// TIA Portal project "practica 9" (V15)

(* hardware
DEVICE "S7-1200 station_1"  S7-1200 Station
   slot 0: "Rack_0"  S7-1200 Rack  Rack  V1.0
   slot 1: "PLC_1"  CPU 1214C AC/DC/Rly  6ES7 214-1BE30-0XB0  V2.2
   slot 3: "AQ 1x12BIT_1"  AQ1 signal board  6ES7 232-4HA30-0XB0  V1.0
DEVICE "S7-1200 station_2"  S7-1200 Station
   slot 0: "Rack_0"  S7-1200 Rack  Rack  V1.0
   slot 1: "PLC_2"  CPU 1214C AC/DC/Rly  6ES7 214-1BG40-0XB0  V4.2
DEVICE "HMI_1"  KTP700 Basic PN
   slot 0: "HMI_1"  KTP700 Basic PN  6AV2 123-2GB03-0AX0  15.0.0.0
   slot 1: "HMI_RT_1"  KTP700 Basic PN  6AV2 123-2GB03-0AX0  15.0.0.0
   slot 5: "HMI_1.IE_CP_1"  PROFINET Interface  15.0.0.0
      slot 1: "Interfaz PROFINET_1"  PROFINET Interface
         slot 1: "Port_1"  Port
*)

// ===== PLC "PLC_1"  CPU 1214C AC/DC/Rly =====

VAR_GLOBAL   // PLC tag table "Tabla de variables estándar"
   "PM" AT %I0.0 : Bool;
   "Paro" AT %I0.1 : Bool;
   "luz verde" AT %Q0.0 : Bool;
   "luz ambar" AT %Q0.1 : Bool;
   "luz roja" AT %Q0.2 : Bool;
   "bucle" AT %M5.0 : Bool;
   "Tag_1" AT %M5.1 : Bool;
   "Luz verde peaton" AT %Q0.4 : Bool;
   "Luz roja peaton" AT %Q0.5 : Bool;
   "Tag_2" AT %M5.2 : Bool;
   "Tag_3" AT %M5.3 : Bool;
END_VAR

// folder: System blocks/Program resources

DATA_BLOCK "IEC_Timer_0_DB"   // DB1
{ S7_Optimized_Access := 'TRUE' }
AUTHOR : Simatic
FAMILY : IEC
NAME : IEC_TMR
VERSION : 1.0
// stored: InstanceOfName IEC_TIMER
"IEC_TIMER"
BEGIN
END_DATA_BLOCK

DATA_BLOCK "IEC_Timer_0_DB_1"   // DB2
{ S7_Optimized_Access := 'TRUE' }
AUTHOR : Simatic
FAMILY : IEC
NAME : IEC_TMR
VERSION : 1.0
// stored: InstanceOfName IEC_TIMER
"IEC_TIMER"
BEGIN
END_DATA_BLOCK

DATA_BLOCK "IEC_Timer_0_DB_2"   // DB3
{ S7_Optimized_Access := 'TRUE' }
AUTHOR : Simatic
FAMILY : IEC
NAME : IEC_TMR
VERSION : 1.0
// stored: InstanceOfName IEC_TIMER
"IEC_TIMER"
BEGIN
END_DATA_BLOCK

DATA_BLOCK "IEC_Timer_0_DB_3"   // DB4
{ S7_Optimized_Access := 'TRUE' }
AUTHOR : Simatic
FAMILY : IEC
NAME : IEC_TMR
VERSION : 1.0
// stored: InstanceOfName IEC_TIMER
"IEC_TIMER"
BEGIN
END_DATA_BLOCK

DATA_BLOCK "IEC_Timer_0_DB_4"   // DB5
{ S7_Optimized_Access := 'TRUE' }
AUTHOR : Simatic
FAMILY : IEC
NAME : IEC_TMR
VERSION : 1.0
// stored: InstanceOfName IEC_TIMER
"IEC_TIMER"
BEGIN
END_DATA_BLOCK

DATA_BLOCK "IEC_Timer_0_DB_5"   // DB6
{ S7_Optimized_Access := 'TRUE' }
AUTHOR : Simatic
FAMILY : IEC
NAME : IEC_TMR
VERSION : 1.0
// stored: InstanceOfName IEC_TIMER
"IEC_TIMER"
BEGIN
END_DATA_BLOCK

DATA_BLOCK "IEC_Timer_0_DB_6"   // DB7
{ S7_Optimized_Access := 'TRUE' }
AUTHOR : Simatic
FAMILY : IEC
NAME : IEC_TMR
VERSION : 1.0
// stored: InstanceOfName IEC_TIMER
"IEC_TIMER"
BEGIN
END_DATA_BLOCK

// folder: (top level)

ORGANIZATION_BLOCK "Main"   // OB1, LAD, ProgramCycle
TITLE = "Main Program Sweep (Cycle)"
{ S7_Optimized_Access := 'TRUE' }
VERSION : 0.1
   VAR_TEMP   // added for the SCL form of the ladder/FBD networks
      _w1 : Bool;
      _w2 : Bool;
   END_VAR
BEGIN

REGION Network 1
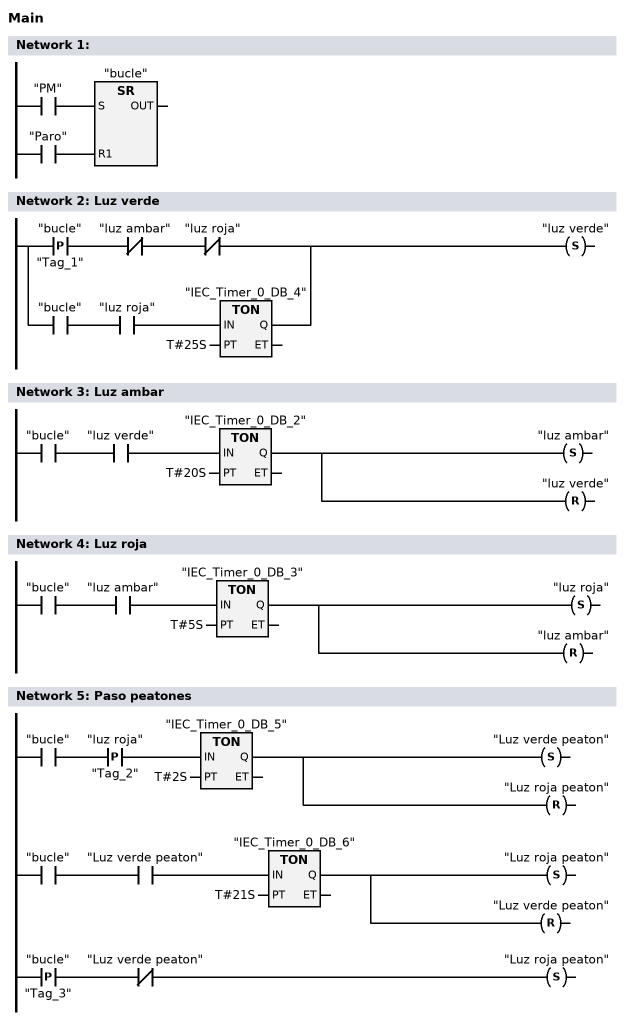
   RUNG wire#powerrail
      Contact( "PM" )
      S_SR(operand := "bucle", r1 := wire#w1)
   END_RUNG
   RUNG wire#powerrail
      Contact( "Paro" )
   END_RUNG wire#w1
   // the same network as SCL:
   IF "PM" THEN
       "bucle" := TRUE;   // SR flip-flop
   END_IF;
   IF "Paro" THEN "bucle" := FALSE; END_IF;
END_REGION

REGION Network 2: Luz verde
   #_w1 := "bucle" AND NOT "Tag_1";   // rising edge of "bucle"
   "Tag_1" := "bucle";
   "IEC_Timer_0_DB_4".TON(IN := "bucle" AND "luz roja", PT := T#25S);
   IF (#_w1 AND NOT "luz ambar" AND NOT "luz roja") OR "IEC_Timer_0_DB_4".Q THEN "luz verde" := TRUE; END_IF;
END_REGION

REGION Network 3: Luz ambar
   "IEC_Timer_0_DB_2".TON(IN := "bucle" AND "luz verde", PT := T#20S);
   IF "IEC_Timer_0_DB_2".Q THEN
       "luz ambar" := TRUE;
       "luz verde" := FALSE;
   END_IF;
END_REGION

REGION Network 4: Luz roja
   "IEC_Timer_0_DB_3".TON(IN := "bucle" AND "luz ambar", PT := T#5S);
   IF "IEC_Timer_0_DB_3".Q THEN
       "luz roja" := TRUE;
       "luz ambar" := FALSE;
   END_IF;
END_REGION

REGION Network 5: Paso peatones
   #_w1 := "bucle" AND "luz roja" AND NOT "Tag_2";   // rising edge of "luz roja"
   "Tag_2" := "luz roja";
   "IEC_Timer_0_DB_5".TON(IN := #_w1, PT := T#2S);
   IF "IEC_Timer_0_DB_5".Q THEN
       "Luz verde peaton" := TRUE;
       "Luz roja peaton" := FALSE;
   END_IF;
   "IEC_Timer_0_DB_6".TON(IN := "bucle" AND "Luz verde peaton", PT := T#21S);
   IF "IEC_Timer_0_DB_6".Q THEN
       "Luz roja peaton" := TRUE;
       "Luz verde peaton" := FALSE;
   END_IF;
   #_w2 := "bucle" AND NOT "Tag_3";   // rising edge of "bucle"
   "Tag_3" := "bucle";
   IF #_w2 AND NOT "Luz verde peaton" THEN "Luz roja peaton" := TRUE; END_IF;
END_REGION

REGION Network 6: Paro peaton
END_REGION
END_ORGANIZATION_BLOCK

// ===== PLC "PLC_2"  CPU 1214C AC/DC/Rly =====

VAR_GLOBAL   // PLC tag table "Tabla de variables estándar"
   "PM" AT %M5.5 : Bool;
   "Paro" AT %I0.1 : Bool;
   "luz verde" AT %Q0.0 : Bool;
   "luz ambar" AT %Q0.1 : Bool;
   "luz roja" AT %Q0.2 : Bool;
   "bucle" AT %M5.0 : Bool;
   "Tag_1" AT %M5.1 : Bool;
   "Luz verde peaton" AT %Q0.4 : Bool;
   "Luz roja peaton" AT %Q0.5 : Bool;
   "Tag_2" AT %M5.2 : Bool;
   "Tag_3" AT %M5.3 : Bool;
   "Clock_Byte" AT %MB256 : Byte;
   "Clock_10Hz" AT %M256.0 : Bool;
   "Clock_5Hz" AT %M256.1 : Bool;
   "Clock_2.5Hz" AT %M256.2 : Bool;
   "Clock_2Hz" AT %M256.3 : Bool;
   "Clock_1.25Hz" AT %M256.4 : Bool;
   "Clock_1Hz" AT %M256.5 : Bool;
   "Clock_0.625Hz" AT %M256.6 : Bool;
   "Clock_0.5Hz" AT %M256.7 : Bool;
   "System_Byte" AT %MB255 : Byte;
   "FirstScan" AT %M255.0 : Bool;
   "DiagStatusUpdate" AT %M255.1 : Bool;
   "AlwaysTRUE" AT %M255.2 : Bool;
   "AlwaysFALSE" AT %M255.3 : Bool;
   "contador" AT %MW258 : Int;
   "Conteo" AT %M6.5 : Bool;
   "Mayor del primer ciclo" AT %M6.6 : Bool;
   "Conteo de ciclos" AT %MW7 : Int;
END_VAR

// folder: System blocks/Program resources

DATA_BLOCK "IEC_Counter_0_DB_1"   // DB1
{ S7_Optimized_Access := 'TRUE' }
AUTHOR : Simatic
FAMILY : IEC
NAME : CNTR
VERSION : 1.0
// stored: InstanceOfName IEC_COUNTER
"IEC_COUNTER"
BEGIN
END_DATA_BLOCK

DATA_BLOCK "IEC_Counter_0_DB"   // DB7
{ S7_Optimized_Access := 'TRUE' }
AUTHOR : Simatic
FAMILY : IEC
NAME : CNTR
VERSION : 1.0
// stored: InstanceOfName IEC_COUNTER
"IEC_COUNTER"
BEGIN
END_DATA_BLOCK

// folder: (top level)

ORGANIZATION_BLOCK "Main"   // OB1, LAD, ProgramCycle
TITLE = "Main Program Sweep (Cycle)"
{ S7_Optimized_Access := 'TRUE' }
VERSION : 0.1
   VAR_INPUT
      Initial_Call : Bool;   // Initial call of this OB
      Remanence : Bool;   // =True, if remanent data are available
   END_VAR
BEGIN

REGION Network 1: Conteo
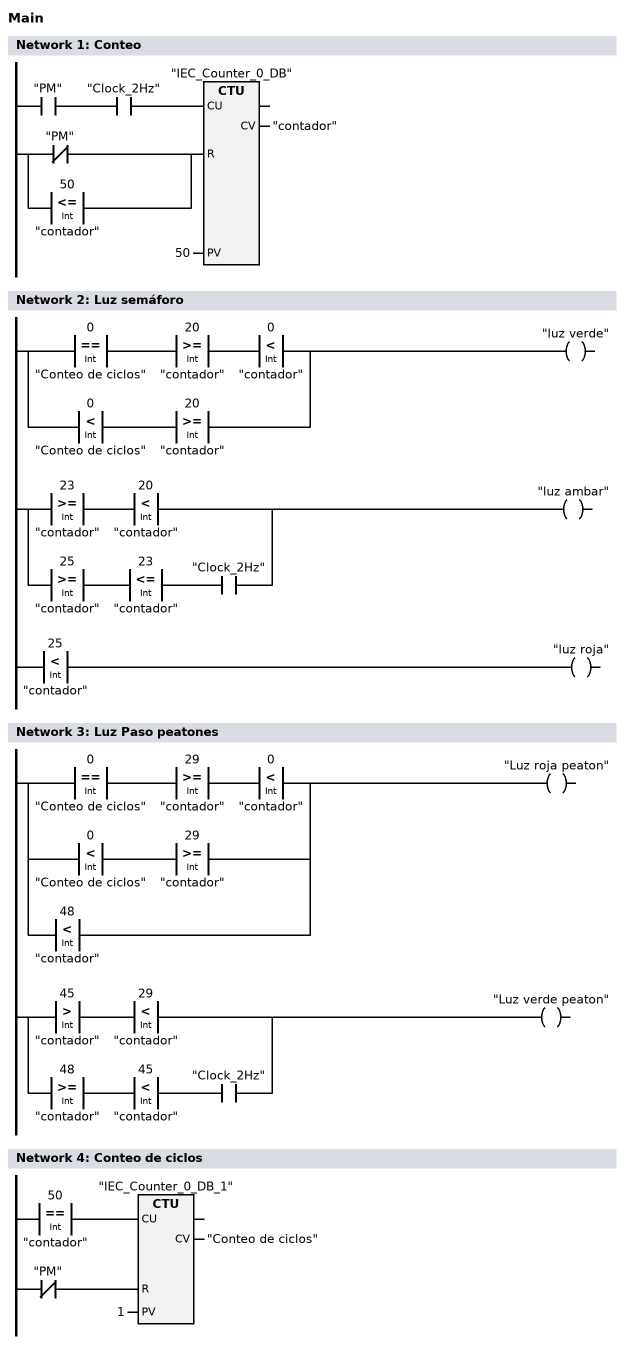
   "IEC_Counter_0_DB".CTU(CU := "PM" AND "Clock_2Hz",
                          R := NOT "PM" OR (50 <= "contador"),
                          PV := 50,
                          CV => "contador");
END_REGION

REGION Network 2: Luz semáforo
   RUNG wire#powerrail
      { S7_Templates := "SrcType := Int" } EQ_Contact(in1 := 0, in2 := "Conteo de ciclos")
      { S7_Templates := "SrcType := Int" } GE_Contact(in1 := 20, in2 := "contador")
      { S7_Templates := "SrcType := Int" } LT_Contact(in1 := 0, in2 := "contador")
      wire#w1
      Coil( "luz verde" )
   END_RUNG
   RUNG wire#powerrail
      { S7_Templates := "SrcType := Int" } LT_Contact(in1 := 0, in2 := "Conteo de ciclos")
      { S7_Templates := "SrcType := Int" } GE_Contact(in1 := 20, in2 := "contador")
   END_RUNG wire#w1
   RUNG wire#powerrail
      { S7_Templates := "SrcType := Int" } GE_Contact(in1 := 23, in2 := "contador")
      { S7_Templates := "SrcType := Int" } LT_Contact(in1 := 20, in2 := "contador")
      wire#w2
      Coil( "luz ambar" )
   END_RUNG
   RUNG wire#powerrail
      { S7_Templates := "SrcType := Int" } GE_Contact(in1 := 25, in2 := "contador")
      { S7_Templates := "SrcType := Int" } LE_Contact(in1 := 23, in2 := "contador")
      Contact( "Clock_2Hz" )
   END_RUNG wire#w2
   RUNG wire#powerrail
      { S7_Templates := "SrcType := Int" } LT_Contact(in1 := 25, in2 := "contador")
      Coil( "luz roja" )
   END_RUNG
   // the same network as SCL:
   "luz verde" := ((0 = "Conteo de ciclos") AND (20 >= "contador") AND (0 < "contador")) OR ((0 < "Conteo de ciclos") AND (20 >= "contador"));
   "luz ambar" := ((23 >= "contador") AND (20 < "contador")) OR ((25 >= "contador") AND (23 <= "contador") AND "Clock_2Hz");
   "luz roja" := 25 < "contador";
END_REGION

REGION Network 3: Luz Paso peatones
   RUNG wire#powerrail
      { S7_Templates := "SrcType := Int" } EQ_Contact(in1 := 0, in2 := "Conteo de ciclos")
      { S7_Templates := "SrcType := Int" } GE_Contact(in1 := 29, in2 := "contador")
      { S7_Templates := "SrcType := Int" } LT_Contact(in1 := 0, in2 := "contador")
      wire#w1
      Coil( "Luz roja peaton" )
   END_RUNG
   RUNG wire#powerrail
      { S7_Templates := "SrcType := Int" } LT_Contact(in1 := 0, in2 := "Conteo de ciclos")
      { S7_Templates := "SrcType := Int" } GE_Contact(in1 := 29, in2 := "contador")
   END_RUNG wire#w1
   RUNG wire#powerrail
      { S7_Templates := "SrcType := Int" } LT_Contact(in1 := 48, in2 := "contador")
   END_RUNG wire#w1
   RUNG wire#powerrail
      { S7_Templates := "SrcType := Int" } GT_Contact(in1 := 45, in2 := "contador")
      { S7_Templates := "SrcType := Int" } LT_Contact(in1 := 29, in2 := "contador")
      wire#w2
      Coil( "Luz verde peaton" )
   END_RUNG
   RUNG wire#powerrail
      { S7_Templates := "SrcType := Int" } GE_Contact(in1 := 48, in2 := "contador")
      { S7_Templates := "SrcType := Int" } LT_Contact(in1 := 45, in2 := "contador")
      Contact( "Clock_2Hz" )
   END_RUNG wire#w2
   // the same network as SCL:
   "Luz roja peaton" := ((0 = "Conteo de ciclos") AND (29 >= "contador") AND (0 < "contador")) OR ((0 < "Conteo de ciclos") AND (29 >= "contador")) OR (48 < "contador");
   "Luz verde peaton" := ((45 > "contador") AND (29 < "contador")) OR ((48 >= "contador") AND (45 < "contador") AND "Clock_2Hz");
END_REGION

REGION Network 4: Conteo de ciclos
   "IEC_Counter_0_DB_1".CTU(CU := 50 = "contador", R := NOT "PM", PV := 1, CV => "Conteo de ciclos");
END_REGION
END_ORGANIZATION_BLOCK

(* ===== HMI "HMI_RT_1" =====
system functions are stored by id; their names below are inferred from use
connection "HMI_Conexión_1": ETHERNET, SMART_S7_1200_OMS

HMI tags "Tabla de variables estándar"
   "Número_imagen_variable" : UInt, internal
   "luz roja" : Bool = PLC "luz roja" AT %Q0.2, 100 ms
   "luz ambar" : Bool = PLC "luz ambar" AT %Q0.1, 100 ms
   "luz verde" : Bool = PLC "luz verde" AT %Q0.0, 100 ms
   "Luz roja peaton" : Bool = PLC "Luz roja peaton" AT %Q0.5, 100 ms
   "Luz verde peaton" : Bool = PLC "Luz verde peaton" AT %Q0.4, 100 ms
   "PM" : Bool = PLC PM AT %M5.5, 1 s

text list "Nombre_imagen_lista_texto": 1 'Imagen raíz'

Template "Plantilla_1" 800x480
   Button "Salir" at 714,429 size 71x50; TextOff 'Salir'; PictureOff "ExitRuntime_KTP700_Basic_PN_TR"; PictureOn "ExitRuntime_KTP700_Basic_PN_TR"
      on Release: StopRuntime(0)
   Button "Template_Button" at 614,429 size 71x50; TextOff 'Text'
   Button "Template_Button_1" at 514,429 size 71x50; TextOff 'Text'
   Button "Template_Button_2" at 414,429 size 71x50; TextOff 'Text'
   Button "Template_Button_3" at 314,429 size 71x50; TextOff 'Text'
   Button "Template_Button_4" at 214,429 size 71x50; TextOff 'Text'
   Button "Avisos" at 114,429 size 71x50; TextOff 'Avisos'; PictureOff "AlarmDisplay_KTP700_Basic_PN_TR"; PictureOn "AlarmDisplay_KTP700_Basic_PN_TR"
      on Release: function_ef3f5d25("Ventana de avisos_no_acusado", -1)
   Button "Imagen inicial" at 14,429 size 71x50; TextOff 'Imagen inicial'; PictureOff "NavigateHome_KTP700_Basic_PN_TR"; PictureOn "NavigateHome_KTP700_Basic_PN_TR"
      on Release: ActivateScreen("Imagen raíz", 0)
   SymbolicIOField "Imagen_campo_ES_simbólico" at 93,9 size 600x33; TextOff '0'; TextOn '1'; TextList "Nombre_imagen_lista_texto"
      ProcessValue <- "Número_imagen_variable"
      on Change: ActivateScreenByNumber("Número_imagen_variable", 0)
   DateTimeField "HmiScreenItemData" at 695,25 size 105x25
   DateTimeField "HmiScreenItemData_1" at 695,0 size 105x25
   GraphicView "Logotipo" at 0,0 size 91x51; Picture "Logotipo de HMI_1"

screen "Imagen raíz" 800x480, template "Plantilla_1"
   on GenerateScreen: SetTag("Número_imagen_variable", 1)
   Circle "Círculo_1" at 132,117 size 68x68
      Appearance <- "luz roja"
   Circle "Círculo_2" at 130,207 size 71x71
      Appearance <- "luz ambar"
   Circle "Círculo_3" at 131,297 size 69x69
      Appearance <- "luz verde"
   Switch "Interruptor_1" at 302,69 size 112x45; CaptionText 'Switch'; TextOff 'OFF'; TextOn 'ON'
      on SwitchOn: SetBit("PM")
      on SwitchOff: ResetBit("PM")
   Circle "Círculo_4" at 499,140 size 76x76
      Appearance <- "Luz roja peaton"
   Circle "Círculo_5" at 499,249 size 76x76
      Appearance <- "Luz verde peaton"
*)